// SIMATIC S7-200 SMART project (STEP 7-Micro/WIN SMART), CPU SR20

SYMBOL_TABLE 表格 1
罗茨清洗定时器          T37
螺杆清洗定时器          T38
吹扫定时器            T39
开机吹扫定时器          T41
开机吹扫定时器2         T42
吹扫定时器2           T43
螺杆清洗定时器2         T44
电流保护延时           T40
延时定时器            T55
流量开关定时器          T56
延时触发             V2.0
DCS_启停指令         VW1106   // 1启动、2停机、3复位、4急停
END_SYMBOL_TABLE

SYMBOL_TABLE 系统符号
Always_On        SM0.0    // 始终接通
First_Scan_On    SM0.1    // 仅在第一个扫描周期时接通
END_SYMBOL_TABLE

SYMBOL_TABLE IO过度V10_30
急停_远程            V10.0    // V10~V30
急停_本地            V10.1    // V10~V30
急停标志位            V10.2    // V10~V30
复位_远程            V10.3    // V10~V30
复位_本地            V10.4    // V10~V30
复位标志位            V10.5    // V10~V30
启动_远程            V10.6    // V10~V30
启动_本地            V10.7    // V10~V30
启动标志位            V11.0    // V10~V30
停机_远程            V11.1    // V10~V30
停机_本地            V11.2    // V10~V30
停机标志位            V11.3    // V10~V30
本地_远程            V11.4    // V10~V30
手动_自动            V11.5    // V10~V30
螺杆泵过载_1          V11.6    // V10~V30
螺杆泵过载_2          V11.7    // V10~V30
螺杆泵过载_3          V12.0    // V10~V30
罗茨泵过载_1          V12.1    // V10~V30
罗茨泵过载_2          V12.2    // V10~V30
罗茨泵过载_3          V12.3    // V10~V30
液环泵过载_1          V12.4    // V10~V30
液环泵过载_2          V12.5    // V10~V30
液环泵过载_3          V12.6    // V10~V30
罗茨冷却风机过载_1       V12.7    // V10~V30
罗茨冷却风机过载_2       V13.0    // V10~V30
罗茨冷却风机过载_3       V13.1    // V10~V30
螺杆冷却风机过载_1       V13.2    // V10~V30
螺杆冷却风机过载_2       V13.3    // V10~V30
螺杆冷却风机过载_3       V13.4    // V10~V30
螺杆变频器故障_1        V13.5    // V10~V30
螺杆变频器故障_2        V13.6    // V10~V30
螺杆变频器故障_3        V13.7    // V10~V30
罗茨变频器故障_1        V14.0    // V10~V30
罗茨变频器故障_2        V14.1    // V10~V30
罗茨变频器故障_3        V14.2    // V10~V30
液环软起动故障_1        V14.3    // V10~V30
液环软起动故障_2        V14.4    // V10~V30
液环软起动故障_3        V14.5    // V10~V30
螺杆流量开关_1         V14.6    // V10~V30
螺杆流量开关_2         V14.7    // V10~V30
螺杆流量开关_3         V15.0    // V10~V30
罗茨流量开关_1         V15.1    // V10~V30
罗茨流量开关_2         V15.2    // V10~V30
罗茨流量开关_3         V15.3    // V10~V30
液环流量开关_1         V15.4    // V10~V30
液环流量开关_2         V15.5    // V10~V30
液环流量开关_3         V15.6    // V10~V30
液位开关_1           V15.7    // V10~V30
液位开关_2           V16.0    // V10~V30
液位开关_3           V16.1    // V10~V30
氮封高压开关           V16.2    // V10~V30
氮封低压开关           V16.3    // V10~V30
真空高压开关           V16.4    // V10~V30
真空低压开关           V16.5    // V10~V30
螺杆泵手动_1          V16.6    // V10~V30
螺杆泵手动_2          V16.7    // V10~V30
螺杆泵手动_3          V17.0    // V10~V30
罗茨泵手动_1          V17.1    // V10~V30
罗茨泵手动_2          V17.2    // V10~V30
罗茨泵手动_3          V17.3    // V10~V30
液环泵手动_1          V17.4    // V10~V30
液环泵手动_2          V17.5    // V10~V30
液环泵手动_3          V17.6    // V10~V30
入口阀手动_1          V17.7    // V10~V30
入口阀手动_2          V18.0    // V10~V30
入口阀手动_3          V18.1    // V10~V30
罗茨清洗阀手动          V18.2    // V10~V30
螺杆清洗阀手动          V18.3    // V10~V30
在线清洗阀手动          V18.4    // V10~V30
吹扫阀手动_1          V18.5    // V10~V30
吹扫阀手动_2          V18.6    // V10~V30
吹扫阀手动_3          V18.7    // V10~V30
进水阀手动_1          V19.0    // V10~V30
进水阀手动_2          V19.1    // V10~V30
进水阀手动_3          V19.2    // V10~V30
排污阀手动_1          V19.3    // V10~V30
排污阀手动_2          V19.4    // V10~V30
排污阀手动_3          V19.5    // V10~V30
螺杆1运行时间清零        V19.6    // V10~V30
螺杆2运行时间清零        V19.7    // V10~V30
故障蜂鸣器            V20.0    // V10~V30
停机指示灯            V20.1    // V10~V30
运行指示灯            V20.2    // V10~V30
清洗吹扫指示灯          V20.3    // V10~V30
螺杆泵_1            V20.4    // V10~V30
螺杆泵_2            V20.5    // V10~V30
螺杆泵_3            V20.6    // V10~V30
罗茨泵_1            V20.7    // V10~V30
罗茨泵_2            V21.0    // V10~V30
罗茨泵_3            V21.1    // V10~V30
液环泵_1            V21.2    // V10~V30
液环泵_2            V21.3    // V10~V30
液环泵_3            V21.4    // V10~V30
入口阀_1            V21.5    // V10~V30
入口阀_2            V21.6    // V10~V30
入口阀_3            V21.7    // V10~V30
罗茨清洗阀            V22.0    // V10~V30
螺杆清洗阀1           V22.1    // V10~V30
在线清洗阀            V22.2    // V10~V30
吹扫阀_1            V22.3    // V10~V30
吹扫阀_2            V22.4    // V10~V30
吹扫阀_3            V22.5    // V10~V30
进水阀_1            V22.6    // V10~V30
进水阀_2            V22.7    // V10~V30
进水阀_3            V23.0    // V10~V30
排污阀_1            V23.1    // V10~V30
排污阀_2            V23.2    // V10~V30
排污阀_3            V23.3    // V10~V30
手动标志位            V23.4    // V10~V30
自动标志位            V23.5    // V10~V30
本地标志位            V23.6    // V10~V30
远程标志位            V23.7    // V10~V30
手动控制_一键复位        V24.0    // V10~V30
故障报警_复位_HMI      V24.1    // HMI指令
入口阀1_开到位         V24.2
入口阀1_关到位         V24.3
入口阀2_开到位         V24.4
入口阀2_关到位         V24.5
螺杆清洗阀2           V24.6
螺杆2清洗阀手动         V24.7
启动_自动_HMI        V25.0    // HMI指令
停机_自动_HMI        V25.1    // HMI指令
手动_自动_HMI        V25.2    // HMI指令
本地_远程_HMI        V25.3    // HMI指令
END_SYMBOL_TABLE

SYMBOL_TABLE ABB_MODUBS
主站完成位            M10.0    // M0~M31
开始轮询             M10.1    // M0~M31
通讯完成位_1          M10.2    // M0~M31
通讯完成位_2          M10.3    // M0~M31
通讯完成位_3          M10.4    // M0~M31
通讯完成位_4          M10.5    // M0~M31
通讯完成位_5          M10.6    // M0~M31
通讯完成位_6          M10.7    // M0~M31
主站_校验            MB4      // 0（无奇偶校验）、1（奇校验）和 2（偶校验）。
主站_端口            MB5      // 0 = CPU 中集成的 RS-485，1 = 可选 CM01 信号板上的 RS-485 或 RS-232
轮询步骤             MB8      // M0~M31
主站故障             MB15     // M0~M31
通讯故障_1           MB16     // M0~M31
通讯故障_2           MB17     // M0~M31
通讯故障_3           MB18     // M0~M31
通讯故障_4           MB19     // M0~M31
通讯故障_5           MB20     // M0~M31
通讯故障_6           MB21     // M0~M31
主站_波特率           MD0      // M0~M31
主站_超时            MW6      // M0~M31
频率写入_1           VB104    // VW100~VW200
频率写入_2           VB110    // VW100~VW200
频率写入_3           VB116    // VW100~VW200
频率读取_1           VW100    // VW100~VW200
电流读取_1           VW102    // VW100~VW200
频率读取_2           VW106    // VW100~VW200
电流读取_2           VW108    // VW100~VW200
频率读取_3           VW112    // VW100~VW200
电流读取_3           VW114    // VW100~VW200
频率显示_1           VW150    // VW100~VW200
电流显示_1           VW152    // VW100~VW200
频率显示_2           VW154    // VW100~VW200
电流显示_2           VW156    // VW100~VW200
频率显示_3           VW158    // VW100~VW200
电流显示_3           VW160    // VW100~VW200
END_SYMBOL_TABLE

SYMBOL_TABLE 故障VW218_222
系统1故障            V217.3
系统2故障            V217.4
A类故障             V217.5
B类故障             V217.6
C类故障             V217.7
A_急停_故障          V218.0
A_螺杆流量开关_故障      V218.1   // VW218-VW222
A_螺杆过载_故障        V218.2   // VW218-VW222
A_氮封低压急停_故障      V218.3   // VW218-VW222
A_螺杆温度急停_故障1     V218.4   // VW218-VW222
A_螺杆变频器_故障1      V218.5   // VW218-VW222
A_螺杆变频器_故障2      V218.6   // VW218-VW222
A_螺杆温度急停_故障2     V218.7   // VW218-VW222
预留_A类故障_3        V219.0   // VW218-VW222
预留_A类故障_4        V219.1   // VW218-VW222
预留_A类故障_5        V219.2   // VW218-VW222
预留_A类故障_6        V219.3   // VW218-VW222
预留_A类故障_7        V219.4   // VW218-VW222
预留_A类故障_8        V219.5   // VW218-VW222
预留_A类故障_9        V219.6   // VW218-VW222
预留_A类故障_10       V219.7   // VW218-VW222
B_罗茨过载1_故障       V220.0   // VW218-VW222
B_罗茨1温度停机_故障     V220.1   // VW218-VW222
B_罗茨过载2_故障       V220.2   // VW218-VW222
B_罗茨2温度停机_故障     V220.3   // VW218-VW222
B_罗茨变频器1_故障      V220.4   // VW218-VW222
B_罗茨变频器2_故障      V220.5   // VW218-VW222
B_罗茨变频器3_故障      V220.6   // VW218-VW222
预留_B类故障_1        V220.7   // VW218-VW222
预留_B类故障_2        V221.0   // VW218-VW222
预留_B类故障_3        V221.1   // VW218-VW222
预留_B类故障_4        V221.2   // VW218-VW222
预留_B类故障_5        V221.3   // VW218-VW222
预留_B类故障_6        V221.4   // VW218-VW222
预留_B类故障_7        V221.5   // VW218-VW222
预留_B类故障_8        V221.6   // VW218-VW222
预留_B类故障_9        V221.7   // VW218-VW222
C_罗茨流量开关_故障      V222.0   // VW218-VW222
C_螺杆温度报警_故障1     V222.1   // VW218-VW222
C_氮封高压报警_故障      V222.2   // VW218-VW222
C_液位过高报警_故障      V222.3   // VW218-VW222
C_罗茨温度报警_故障      V222.4   // VW218-VW222
C_螺杆温度报警_故障2     V222.5   // VW218-VW222
预留_C类故障_2        V222.6   // VW218-VW222
预留_C类故障_3        V222.7   // VW218-VW222
预留_C类故障_4        V223.0   // VW218-VW222
预留_C类故障_5        V223.1   // VW218-VW222
预留_C类故障_6        V223.2   // VW218-VW222
预留_C类故障_7        V223.3   // VW218-VW222
预留_C类故障_8        V223.4   // VW218-VW222
预留_C类故障_9        V223.5   // VW218-VW222
预留_C类故障_10       V223.6   // VW218-VW222
预留_C类故障_11       V223.7   // VW218-VW222
END_SYMBOL_TABLE

SYMBOL_TABLE 参数设置VW1000_1148
罗茨_温度报警_设置       VD1000   // VW1000~VW1148
罗茨_温度停机_设置       VD1004   // VW1000~VW1148
液位_过高报警_设置       VD1008   // VW1000~VW1148
螺杆_温度报警_设置       VD1012   // VW1000~VW1148
螺杆_温度停机_设置       VD1016   // VW1000~VW1148
电流_保护_设置         VD1020   // VW1000~VW1148
电流_恢复_设置         VD1024   // VW1000~VW1148
液位_保护_设置         VD1028   // VW1000~VW1148
液位_恢复_设置         VD1032   // VW1000~VW1148
液位_变送器上限_设置      VD1036   // VW1000~VW1148
螺杆温度_变送器上限_设     VD1040   // VW1000~VW1148
电流_变送器上限_设置      VD1044   // VW1000~VW1148
罗茨1温度_变送器上限_设    VD1048   // VW1000~VW1148
罗茨2温度_变送器上限_设    VD1052   // VW1000~VW1148
罗茨1启动真空设定        VD1056   // VW1000~VW1148
罗茨1停机真空设定        VD1060   // VW1000~VW1148
罗茨2启动真空设定        VD1064   // VW1000~VW1148
罗茨2停机真空设定        VD1068   // VW1000~VW1148
真空_变送器上限_设定      VD1072   // VW1000~VW1148
氮气_变送器上限_设定      VD1076   // VW1000~VW1148
氮气_低压急停_设定       VD1080   // VW1000~VW1148
氮气_低压报警_设定       VD1084   // VW1000~VW1148
目标真空度_设定         VD1088   // VW1000~VW1148
                 VD1092   // VW1000~VW1148
                 VD1096   // VW1000~VW1148
DCS_校验_设置        VD1144   // VW1000~VW1148
罗茨_清洗时间_设置       VW1100   // VW1000~VW1148
螺杆_清洗时间_设置       VW1102   // VW1000~VW1148
吹扫_时间_设置         VW1104   // VW1000~VW1148
螺杆手动频率_设置        VW1108   // VW1000~VW1148
罗茨1手动频率_设置       VW1110   // VW1000~VW1148
罗茨2手动频率_设置       VW1112   // VW1000~VW1148
螺杆清洗频率_设置        VW1114   // VW1000~VW1148
螺杆2手动频率_设置       VW1116   // VW1000~VW1148
螺杆2清洗频率_设置       VW1118   // VW1000~VW1148
开机吹扫_时间_设置       VW1120   // VW1000~VW1148
电流过载_预防_设置       VW1122   // VW1000~VW1148
                 VW1124   // VW1000~VW1148
                 VW1126   // VW1000~VW1148
                 VW1128   // VW1000~VW1148
                 VW1130   // VW1000~VW1148
                 VW1132   // VW1000~VW1148
                 VW1134   // VW1000~VW1148
                 VW1136   // VW1000~VW1148
                 VW1138   // VW1000~VW1148
DCS_地址_设置        VW1140   // VW1000~VW1148
DCS_波特率_设置       VW1142   // VW1000~VW1148
                 VW1148   // VW1000~VW1148
                          // VW1000~VW1148
END_SYMBOL_TABLE

SYMBOL_TABLE 参数显示
螺杆温度值1           VD1154
罗茨液位值            VD1158
螺杆液位值            VD1162
螺杆电流值            VD1166
机组真空度            VD1170
罗茨温度值            VD1178
绝对真空显示           VD1182
自动步骤1            VW1202
自动步骤2            VW1204
开机吹扫_时间_显示       VW1206
螺杆_清洗时间_显示       VW1208
罗茨_清洗时间_显示       VW1210
吹扫时间_显示          VW1212
螺杆_频率_显示         VW1214
螺杆_电流_显示         VW1216
罗茨1_频率_显示        VW1218
罗茨1_电流_显示        VW1220
罗茨2_频率_显示        VW1222
罗茨2_电流_显示        VW1224
螺杆1运行时间_秒        VW1226
螺杆1运行时间_分        VW1228
螺杆1运行时间_时        VW1230
螺杆2运行时间_秒        VW1232
螺杆2运行时间_分        VW1234
螺杆2运行时间_时        VW1236
螺杆温度值2           VD1186
螺杆温度值3           VD1190
入口温度1            VD1194
入口温度2            VD1198
螺杆2_频率_显示        VW1238
螺杆2_电流_显示        VW1240
END_SYMBOL_TABLE

SYMBOL_TABLE 变送器VD30_96
真空变送器            VW30     // VD30~VD96
螺杆温度变送器_1        VW32     // VD30~VD96
螺杆温度变送器_2        VW34     // VD30~VD96
螺杆温度变送器_3        VW36     // VD30~VD96
罗茨温度变送器_1        VW38     // VD30~VD96
罗茨温度变送器_2        VW40     // VD30~VD96
罗茨温度变送器_3        VW42     // VD30~VD96
液环温度变送器_1        VW44     // VD30~VD96
液环温度变送器_2        VW46     // VD30~VD96
液环温度变送器_3        VW48     // VD30~VD96
入口温度变送器1         VW50     // VD30~VD96
液位变送器            VW52     // VD30~VD96
前端液位变送器          VW54     // VD30~VD96
后端液位变送器          VW56     // VD30~VD96
螺杆电流变送器          VW58     // VD30~VD96
入口温度变送器2         VW60     // VD30~VD96
END_SYMBOL_TABLE

SYMBOL_TABLE 辅助点表
急停_远程_使能         V300.0
急停_本地_使能         V300.1
急停标志位_使能         V300.2
复位_远程_使能         V300.3
复位_本地_使能         V300.4
复位标志位_使能         V300.5
启动_远程_使能         V300.6
启动_本地_使能         V300.7
启动标志位_使能         V301.0
停机_远程_使能         V301.1
停机_本地_使能         V301.2
停机标志位_使能         V301.3
本地_远程_使能         V301.4
手动_自动_使能         V301.5
螺杆泵过载_1_使能       V301.6
螺杆泵过载_2_使能       V301.7
螺杆泵过载_3_使能       V302.0
罗茨泵过载_1_使能       V302.1
罗茨泵过载_2_使能       V302.2
罗茨泵过载_3_使能       V302.3
液环泵过载_1_使能       V302.4
液环泵过载_2_使能       V302.5
液环泵过载_3_使能       V302.6
罗茨冷却风机过载_1_使能    V302.7
罗茨冷却风机过载_2_使能    V303.0
罗茨冷却风机过载_3_使能    V303.1
螺杆冷却风机过载_1_使能    V303.2
螺杆冷却风机过载_2_使能    V303.3
螺杆冷却风机过载_3_使能    V303.4
螺杆变频器故障_1_使能     V303.5
螺杆变频器故障_2_使能     V303.6
螺杆变频器故障_3_使能     V303.7
罗茨变频器故障_1_使能     V304.0
罗茨变频器故障_2_使能     V304.1
罗茨变频器故障_3_使能     V304.2
液环软起动故障_1_使能     V304.3
液环软起动故障_2_使能     V304.4
液环软起动故障_3_使能     V304.5
螺杆流量开关_1_使能      V304.6
螺杆流量开关_2_使能      V304.7
螺杆流量开关_3_使能      V305.0
罗茨流量开关_1_使能      V305.1
罗茨流量开关_2_使能      V305.2
罗茨流量开关_3_使能      V305.3
液环流量开关_1_使能      V305.4
液环流量开关_2_使能      V305.5
液环流量开关_3_使能      V305.6
液位开关_1_使能        V305.7
液位开关_2_使能        V306.0
液位开关_3_使能        V306.1
氮封高压开关_使能        V306.2
氮封低压开关_使能        V306.3
真空高压开关_使能        V306.4
真空低压开关_使能        V306.5
螺杆泵手动_1_使能       V306.6
螺杆泵手动_2_使能       V306.7
螺杆泵手动_3_使能       V307.0
罗茨泵手动_1_使能       V307.1
罗茨泵手动_2_使能       V307.2
罗茨泵手动_3_使能       V307.3
液环泵手动_1_使能       V307.4
液环泵手动_2_使能       V307.5
液环泵手动_3_使能       V307.6
入口阀手动_1_使能       V307.7
入口阀手动_2_使能       V308.0
入口阀手动_3_使能       V308.1
罗茨清洗阀手动_使能       V308.2
螺杆1清洗阀手动_使能      V308.3
在线清洗阀手动_使能       V308.4
吹扫阀手动_1_使能       V308.5
吹扫阀手动_2_使能       V308.6
吹扫阀手动_3_使能       V308.7
进水阀手动_1_使能       V309.0
进水阀手动_2_使能       V309.1
进水阀手动_3_使能       V309.2
排污阀手动_1_使能       V309.3
排污阀手动_2_使能       V309.4
排污阀手动_3_使能       V309.5
螺杆1运行时间清零_使能     V309.6
螺杆2运行时间清零_使能     V309.7
故障蜂鸣器_使能         V310.0
停机指示灯_使能         V310.1
运行指示灯_使能         V310.2
清洗吹扫指示灯_使能       V310.3
螺杆泵_1_使能         V310.4
螺杆泵_2_使能         V310.5
螺杆泵_3_使能         V310.6
罗茨泵_1_使能         V310.7
罗茨泵_2_使能         V311.0
罗茨泵_3_使能         V311.1
液环泵_1_使能         V311.2
液环泵_2_使能         V311.3
液环泵_3_使能         V311.4
入口阀_1_使能         V311.5
入口阀_2_使能         V311.6
入口阀_3_使能         V311.7
罗茨清洗阀_使能         V312.0
螺杆清洗阀1_使能        V312.1
在线清洗阀_使能         V312.2
吹扫阀_1_使能         V312.3
吹扫阀_2_使能         V312.4
吹扫阀_3_使能         V312.5
进水阀_1_使能         V312.6
进水阀_2_使能         V312.7
进水阀_3_使能         V313.0
排污阀_1_使能         V313.1
排污阀_2_使能         V313.2
排污阀_3_使能         V313.3
手动标志位_使能         V313.4
自动标志位_使能         V313.5
本地标志位_使能         V313.6
远程标志位_使能         V313.7
手动控制_一键复位_使能     V314.0
故障报警_复位_HMI_使能   V314.1
入口阀1_开到位_使能      V314.2
入口阀1_关到位_使能      V314.3
入口阀2_开到位_使能      V314.4
入口阀2_关到位_使能      V314.5
螺杆清洗阀2_使能        V314.6
系统1_使能           V315.0
系统2_使能           V315.1
系统3_使能           V315.2
优先启动机组           V315.3
螺杆2清洗阀手动_使能      V314.7
END_SYMBOL_TABLE

SYMBOL_TABLE 中间变量
开机吹扫_时间_中间值      VW5000
吹扫_时间_中间值        VW5002
螺杆_清洗时间_中间值      VW5004
罗茨_清洗时间_中间值      VW5006
PID_频率1          VW5008
PID_频率2          VW5010
END_SYMBOL_TABLE

SYMBOL_TABLE PID数据
PID故障1           VB5200
PID故障2           VB5201
END_SYMBOL_TABLE

ORGANIZATION_BLOCK MAIN:OB1
TITLE=程序注释
BEGIN
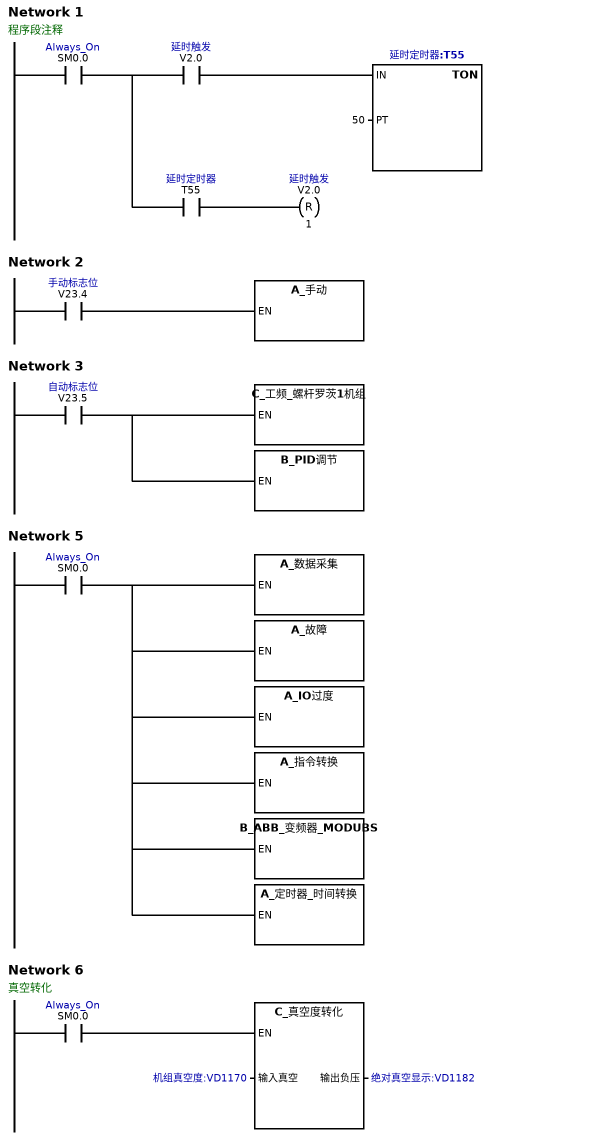
Network 1
// 程序段注释
LD     Always_On:SM0.0
LPS
A      延时触发:V2.0
TON    延时定时器:T55, 50
LPP
A      延时定时器:T55
R      延时触发:V2.0, 1
Network 2
LD     手动标志位:V23.4
CALL   A_手动:SBR0
Network 3
LD     自动标志位:V23.5
CALL   C_工频_螺杆罗茨1机组:SBR1
CALL   B_PID调节:SBR22
Network 5
LD     Always_On:SM0.0
CALL   A_数据采集:SBR2
CALL   A_故障:SBR3
CALL   A_IO过度:SBR5
CALL   A_指令转换:SBR11
CALL   B_ABB_变频器_MODUBS:SBR7
CALL   A_定时器_时间转换:SBR21
Network 6
// 真空转化
LD     Always_On:SM0.0
CALL   C_真空度转化:SBR12, 机组真空度:VD1170, 绝对真空显示:VD1182
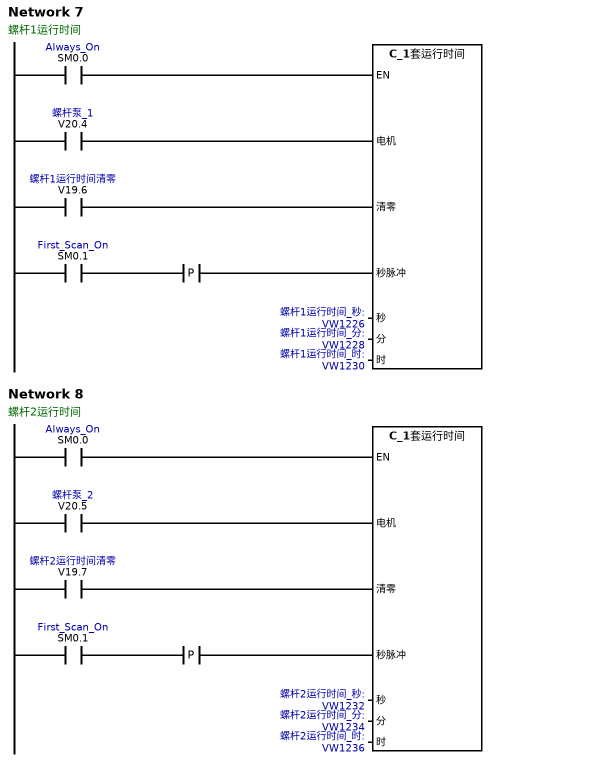
Network 7
// 螺杆1运行时间
LD     Always_On:SM0.0
=      L60.0
LD     螺杆泵_1:V20.4
=      L63.7
LD     螺杆1运行时间清零:V19.6
=      L63.6
LD     First_Scan_On:SM0.1
EU
=      L63.5
LD     L60.0
CALL   C_1套运行时间:SBR13, L63.7, L63.6, L63.5, 螺杆1运行时间_秒:VW1226, 螺杆1运行时间_分:VW1228, 螺杆1运行时间_时:VW1230
Network 8
// 螺杆2运行时间
LD     Always_On:SM0.0
=      L60.0
LD     螺杆泵_2:V20.5
=      L63.7
LD     螺杆2运行时间清零:V19.7
=      L63.6
LD     First_Scan_On:SM0.1
EU
=      L63.5
LD     L60.0
CALL   C_1套运行时间:SBR13, L63.7, L63.6, L63.5, 螺杆2运行时间_秒:VW1232, 螺杆2运行时间_分:VW1234, 螺杆2运行时间_时:VW1236
END_ORGANIZATION_BLOCK

SUBROUTINE_BLOCK A_手动:SBR0
TITLE=子程序注释
BEGIN
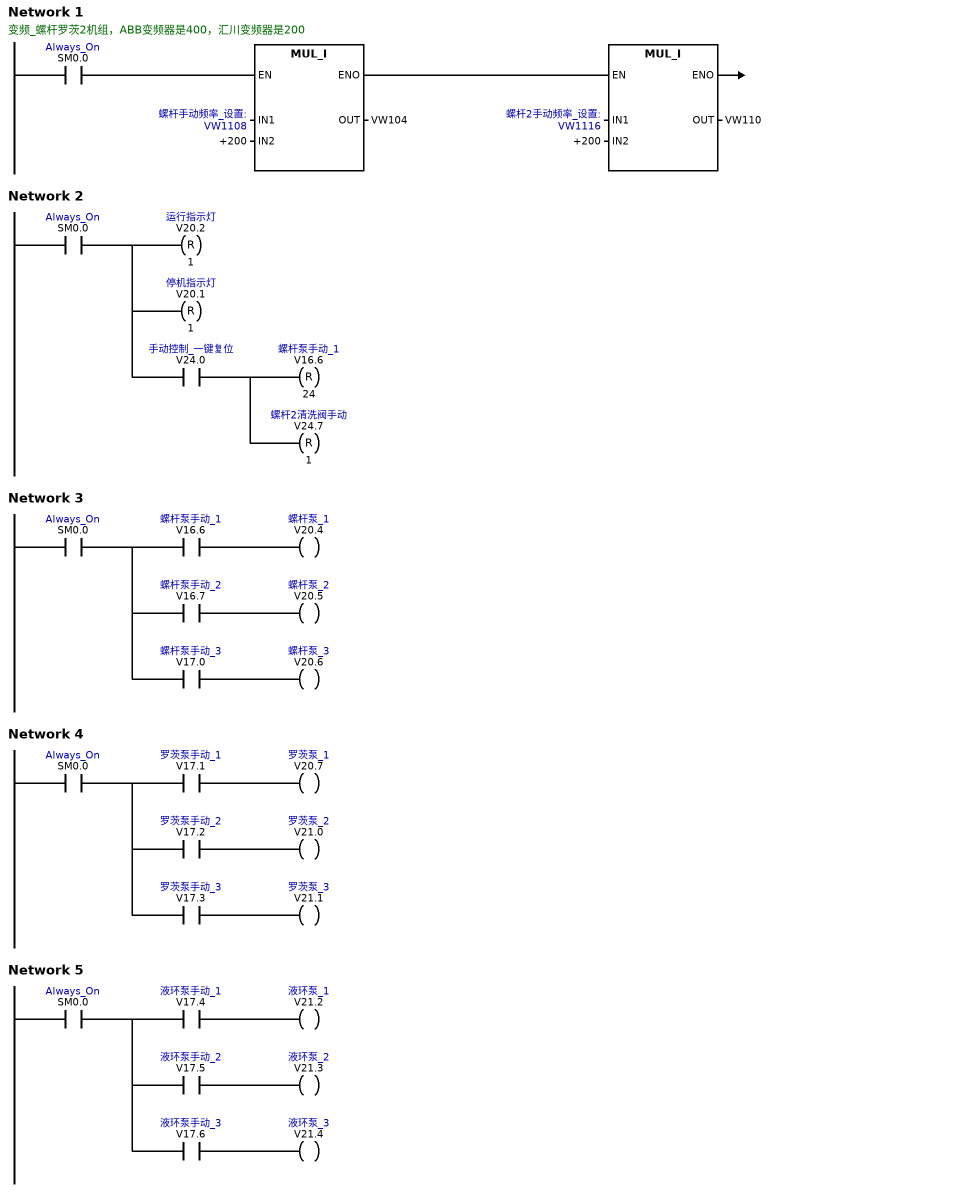
Network 1
// 变频_螺杆罗茨2机组，ABB变频器是400，汇川变频器是200
LD     Always_On:SM0.0
MOVW   螺杆手动频率_设置:VW1108, VW104
AENO
*I     +200, VW104
AENO
MOVW   螺杆2手动频率_设置:VW1116, VW110
*I     +200, VW110
Network 2
LD     Always_On:SM0.0
R      运行指示灯:V20.2, 1
R      停机指示灯:V20.1, 1
A      手动控制_一键复位:V24.0
R      螺杆泵手动_1:V16.6, 24
R      螺杆2清洗阀手动:V24.7, 1
Network 3
LD     Always_On:SM0.0
LPS
A      螺杆泵手动_1:V16.6
=      螺杆泵_1:V20.4
LRD
A      螺杆泵手动_2:V16.7
=      螺杆泵_2:V20.5
LPP
A      螺杆泵手动_3:V17.0
=      螺杆泵_3:V20.6
Network 4
LD     Always_On:SM0.0
LPS
A      罗茨泵手动_1:V17.1
=      罗茨泵_1:V20.7
LRD
A      罗茨泵手动_2:V17.2
=      罗茨泵_2:V21.0
LPP
A      罗茨泵手动_3:V17.3
=      罗茨泵_3:V21.1
Network 5
LD     Always_On:SM0.0
LPS
A      液环泵手动_1:V17.4
=      液环泵_1:V21.2
LRD
A      液环泵手动_2:V17.5
=      液环泵_2:V21.3
LPP
A      液环泵手动_3:V17.6
=      液环泵_3:V21.4
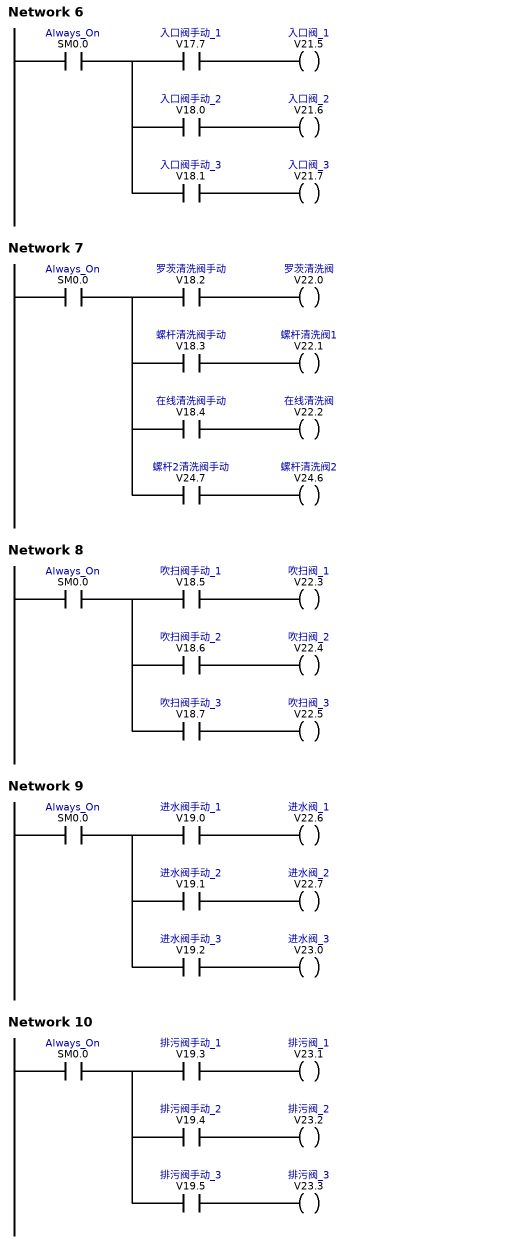
Network 6
LD     Always_On:SM0.0
LPS
A      入口阀手动_1:V17.7
=      入口阀_1:V21.5
LRD
A      入口阀手动_2:V18.0
=      入口阀_2:V21.6
LPP
A      入口阀手动_3:V18.1
=      入口阀_3:V21.7
Network 7
LD     Always_On:SM0.0
LPS
A      罗茨清洗阀手动:V18.2
=      罗茨清洗阀:V22.0
LRD
A      螺杆清洗阀手动:V18.3
=      螺杆清洗阀1:V22.1
LRD
A      在线清洗阀手动:V18.4
=      在线清洗阀:V22.2
LPP
A      螺杆2清洗阀手动:V24.7
=      螺杆清洗阀2:V24.6
Network 8
LD     Always_On:SM0.0
LPS
A      吹扫阀手动_1:V18.5
=      吹扫阀_1:V22.3
LRD
A      吹扫阀手动_2:V18.6
=      吹扫阀_2:V22.4
LPP
A      吹扫阀手动_3:V18.7
=      吹扫阀_3:V22.5
Network 9
LD     Always_On:SM0.0
LPS
A      进水阀手动_1:V19.0
=      进水阀_1:V22.6
LRD
A      进水阀手动_2:V19.1
=      进水阀_2:V22.7
LPP
A      进水阀手动_3:V19.2
=      进水阀_3:V23.0
Network 10
LD     Always_On:SM0.0
LPS
A      排污阀手动_1:V19.3
=      排污阀_1:V23.1
LRD
A      排污阀手动_2:V19.4
=      排污阀_2:V23.2
LPP
A      排污阀手动_3:V19.5
=      排污阀_3:V23.3
END_SUBROUTINE_BLOCK

SUBROUTINE_BLOCK C_工频_螺杆罗茨1机组:SBR1
TITLE=子程序注释
BEGIN
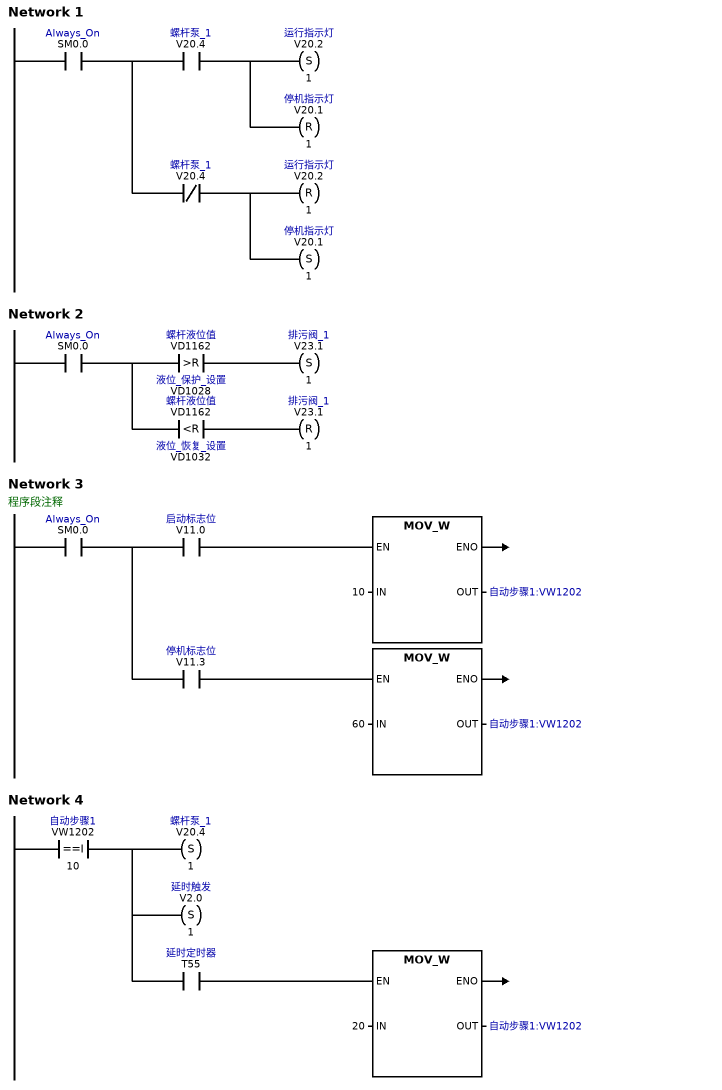
Network 1
LD     Always_On:SM0.0
LPS
A      螺杆泵_1:V20.4
S      运行指示灯:V20.2, 1
R      停机指示灯:V20.1, 1
LPP
AN     螺杆泵_1:V20.4
R      运行指示灯:V20.2, 1
S      停机指示灯:V20.1, 1
Network 2
LD     Always_On:SM0.0
LPS
AR>    螺杆液位值:VD1162, 液位_保护_设置:VD1028
S      排污阀_1:V23.1, 1
LPP
AR<    螺杆液位值:VD1162, 液位_恢复_设置:VD1032
R      排污阀_1:V23.1, 1
Network 3
// 程序段注释
LD     Always_On:SM0.0
LPS
A      启动标志位:V11.0
MOVW   10, 自动步骤1:VW1202
LPP
A      停机标志位:V11.3
MOVW   60, 自动步骤1:VW1202
Network 4
LDW=   自动步骤1:VW1202, 10
S      螺杆泵_1:V20.4, 1
S      延时触发:V2.0, 1
A      延时定时器:T55
MOVW   20, 自动步骤1:VW1202
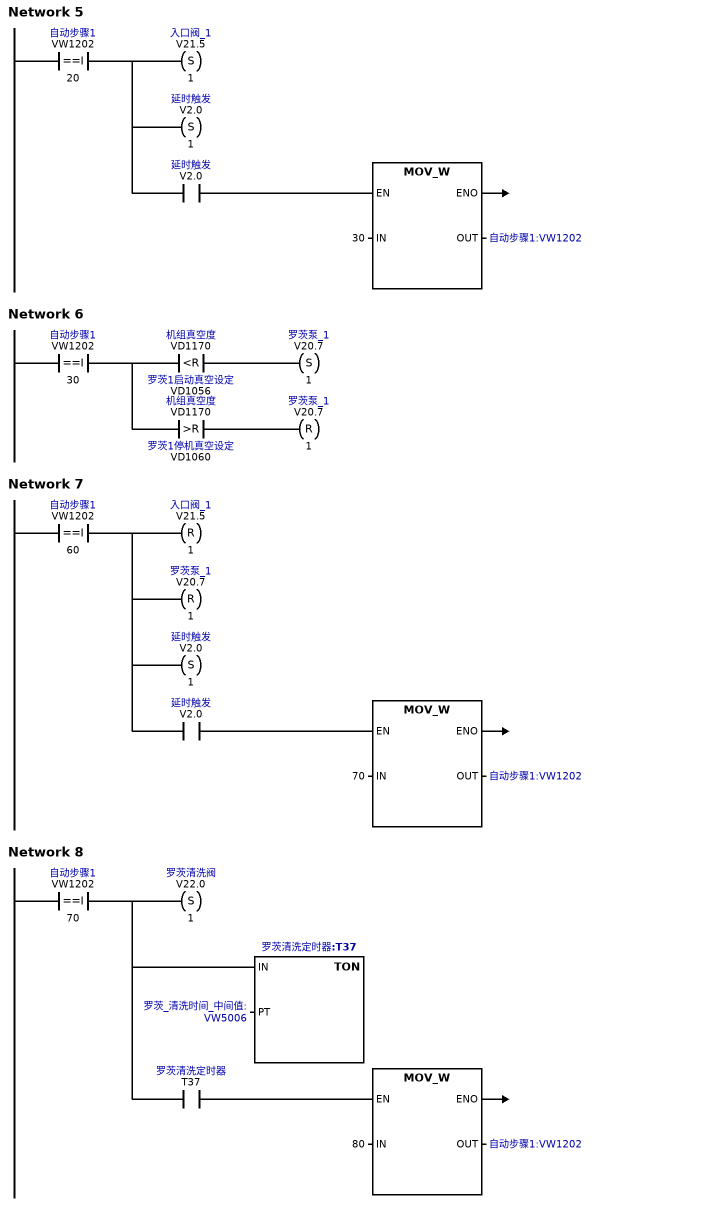
Network 5
LDW=   自动步骤1:VW1202, 20
S      入口阀_1:V21.5, 1
S      延时触发:V2.0, 1
A      延时触发:V2.0
MOVW   30, 自动步骤1:VW1202
Network 6
LDW=   自动步骤1:VW1202, 30
LPS
AR<    机组真空度:VD1170, 罗茨1启动真空设定:VD1056
S      罗茨泵_1:V20.7, 1
LPP
AR>    机组真空度:VD1170, 罗茨1停机真空设定:VD1060
R      罗茨泵_1:V20.7, 1
Network 7
LDW=   自动步骤1:VW1202, 60
R      入口阀_1:V21.5, 1
R      罗茨泵_1:V20.7, 1
S      延时触发:V2.0, 1
A      延时触发:V2.0
MOVW   70, 自动步骤1:VW1202
Network 8
LDW=   自动步骤1:VW1202, 70
S      罗茨清洗阀:V22.0, 1
TON    罗茨清洗定时器:T37, 罗茨_清洗时间_中间值:VW5006
A      罗茨清洗定时器:T37
MOVW   80, 自动步骤1:VW1202
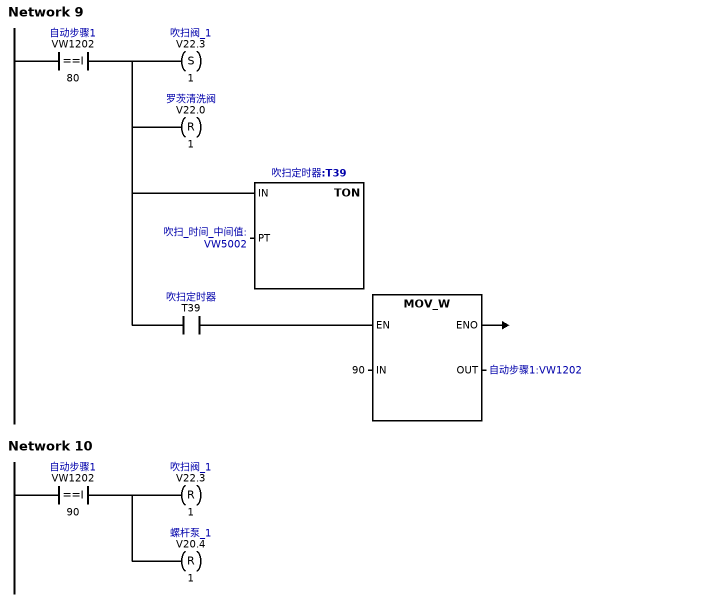
Network 9
LDW=   自动步骤1:VW1202, 80
S      吹扫阀_1:V22.3, 1
R      罗茨清洗阀:V22.0, 1
TON    吹扫定时器:T39, 吹扫_时间_中间值:VW5002
A      吹扫定时器:T39
MOVW   90, 自动步骤1:VW1202
Network 10
LDW=   自动步骤1:VW1202, 90
R      吹扫阀_1:V22.3, 1
R      螺杆泵_1:V20.4, 1
END_SUBROUTINE_BLOCK

SUBROUTINE_BLOCK A_数据采集:SBR2
TITLE=子程序注释
BEGIN
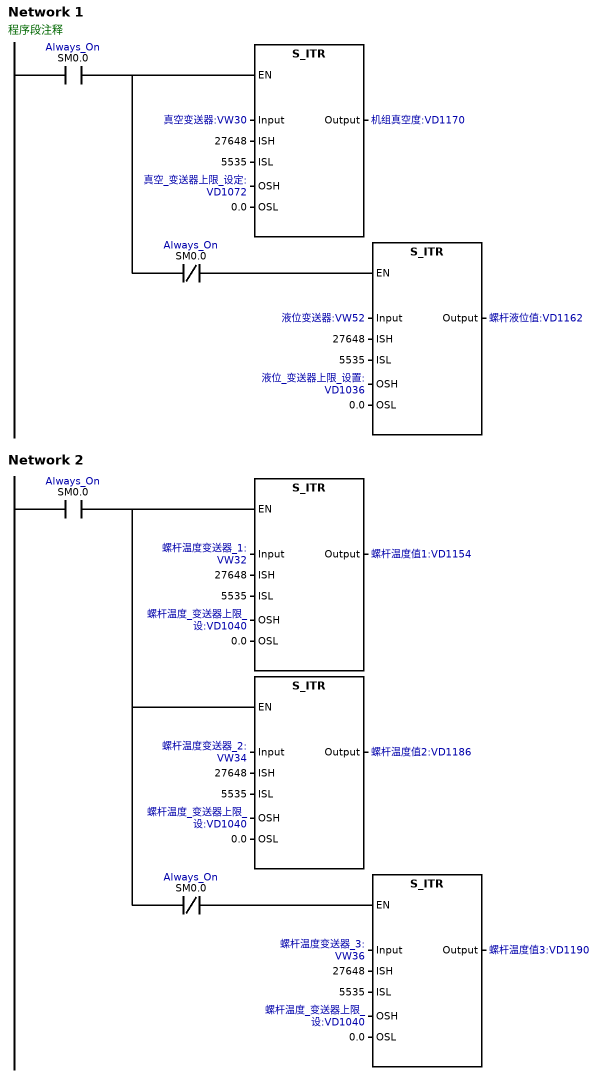
Network 1
// 程序段注释
LD     Always_On:SM0.0
CALL   S_ITR:SBR4, 真空变送器:VW30, 27648, 5535, 真空_变送器上限_设定:VD1072, 0.0, 机组真空度:VD1170
AN     Always_On:SM0.0
CALL   S_ITR:SBR4, 液位变送器:VW52, 27648, 5535, 液位_变送器上限_设置:VD1036, 0.0, 螺杆液位值:VD1162
Network 2
LD     Always_On:SM0.0
CALL   S_ITR:SBR4, 螺杆温度变送器_1:VW32, 27648, 5535, 螺杆温度_变送器上限_设:VD1040, 0.0, 螺杆温度值1:VD1154
CALL   S_ITR:SBR4, 螺杆温度变送器_2:VW34, 27648, 5535, 螺杆温度_变送器上限_设:VD1040, 0.0, 螺杆温度值2:VD1186
AN     Always_On:SM0.0
CALL   S_ITR:SBR4, 螺杆温度变送器_3:VW36, 27648, 5535, 螺杆温度_变送器上限_设:VD1040, 0.0, 螺杆温度值3:VD1190
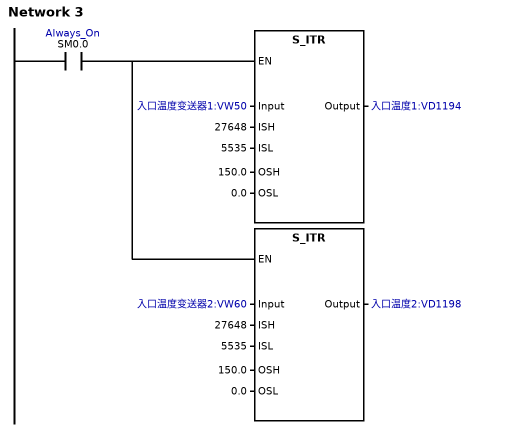
Network 3
LD     Always_On:SM0.0
CALL   S_ITR:SBR4, 入口温度变送器1:VW50, 27648, 5535, 150.0, 0.0, 入口温度1:VD1194
CALL   S_ITR:SBR4, 入口温度变送器2:VW60, 27648, 5535, 150.0, 0.0, 入口温度2:VD1198
END_SUBROUTINE_BLOCK

SUBROUTINE_BLOCK A_故障:SBR3
TITLE=子程序注释
BEGIN
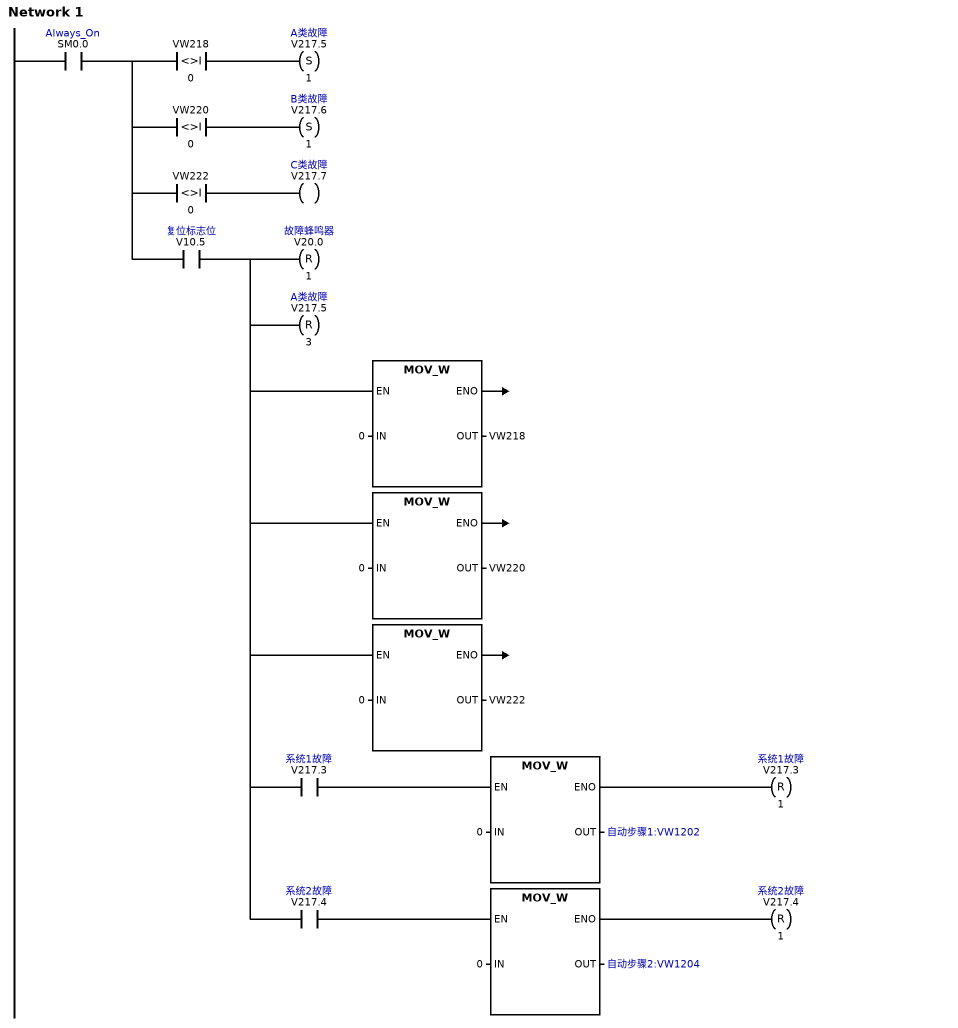
Network 1
LD     Always_On:SM0.0
LPS
AW<>   VW218, 0
S      A类故障:V217.5, 1
LRD
AW<>   VW220, 0
S      B类故障:V217.6, 1
LRD
AW<>   VW222, 0
=      C类故障:V217.7
LPP
A      复位标志位:V10.5
LPS
R      故障蜂鸣器:V20.0, 1
R      A类故障:V217.5, 3
MOVW   0, VW218
MOVW   0, VW220
MOVW   0, VW222
A      系统1故障:V217.3
MOVW   0, 自动步骤1:VW1202
AENO
R      系统1故障:V217.3, 1
LPP
A      系统2故障:V217.4
MOVW   0, 自动步骤2:VW1204
AENO
R      系统2故障:V217.4, 1
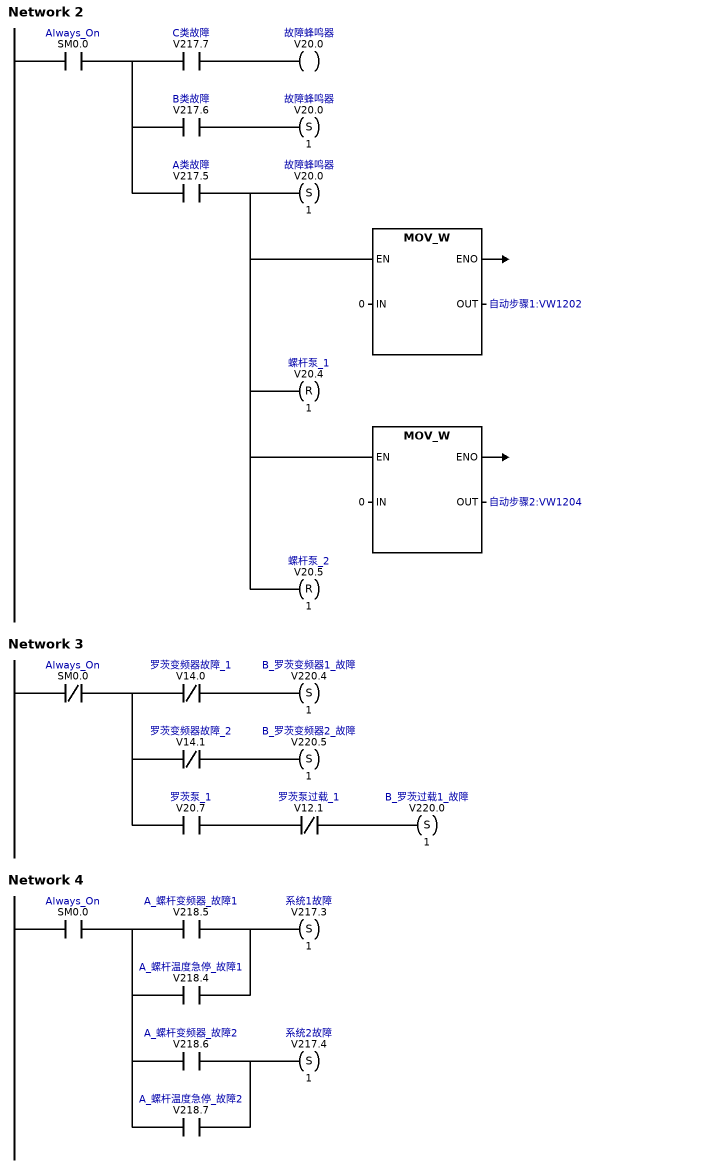
Network 2
LD     Always_On:SM0.0
LPS
A      C类故障:V217.7
=      故障蜂鸣器:V20.0
LRD
A      B类故障:V217.6
S      故障蜂鸣器:V20.0, 1
LPP
A      A类故障:V217.5
S      故障蜂鸣器:V20.0, 1
MOVW   0, 自动步骤1:VW1202
R      螺杆泵_1:V20.4, 1
MOVW   0, 自动步骤2:VW1204
R      螺杆泵_2:V20.5, 1
Network 3
LDN    Always_On:SM0.0
LPS
AN     罗茨变频器故障_1:V14.0
S      B_罗茨变频器1_故障:V220.4, 1
LRD
AN     罗茨变频器故障_2:V14.1
S      B_罗茨变频器2_故障:V220.5, 1
LPP
A      罗茨泵_1:V20.7
AN     罗茨泵过载_1:V12.1
S      B_罗茨过载1_故障:V220.0, 1
Network 4
LD     Always_On:SM0.0
LPS
LD     A_螺杆变频器_故障1:V218.5
O      A_螺杆温度急停_故障1:V218.4
ALD
S      系统1故障:V217.3, 1
LPP
LD     A_螺杆变频器_故障2:V218.6
O      A_螺杆温度急停_故障2:V218.7
ALD
S      系统2故障:V217.4, 1
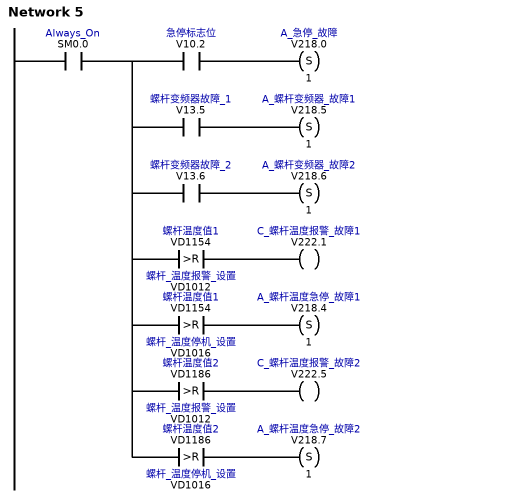
Network 5
LD     Always_On:SM0.0
LPS
A      急停标志位:V10.2
S      A_急停_故障:V218.0, 1
LRD
A      螺杆变频器故障_1:V13.5
S      A_螺杆变频器_故障1:V218.5, 1
LRD
A      螺杆变频器故障_2:V13.6
S      A_螺杆变频器_故障2:V218.6, 1
LRD
AR>    螺杆温度值1:VD1154, 螺杆_温度报警_设置:VD1012
=      C_螺杆温度报警_故障1:V222.1
LRD
AR>    螺杆温度值1:VD1154, 螺杆_温度停机_设置:VD1016
S      A_螺杆温度急停_故障1:V218.4, 1
LRD
AR>    螺杆温度值2:VD1186, 螺杆_温度报警_设置:VD1012
=      C_螺杆温度报警_故障2:V222.5
LPP
AR>    螺杆温度值2:VD1186, 螺杆_温度停机_设置:VD1016
S      A_螺杆温度急停_故障2:V218.7, 1
END_SUBROUTINE_BLOCK

// SBR4: protected block, not included

SUBROUTINE_BLOCK A_IO过度:SBR5
TITLE=DI,DO,AI,AO过渡，占用V10~100
BEGIN
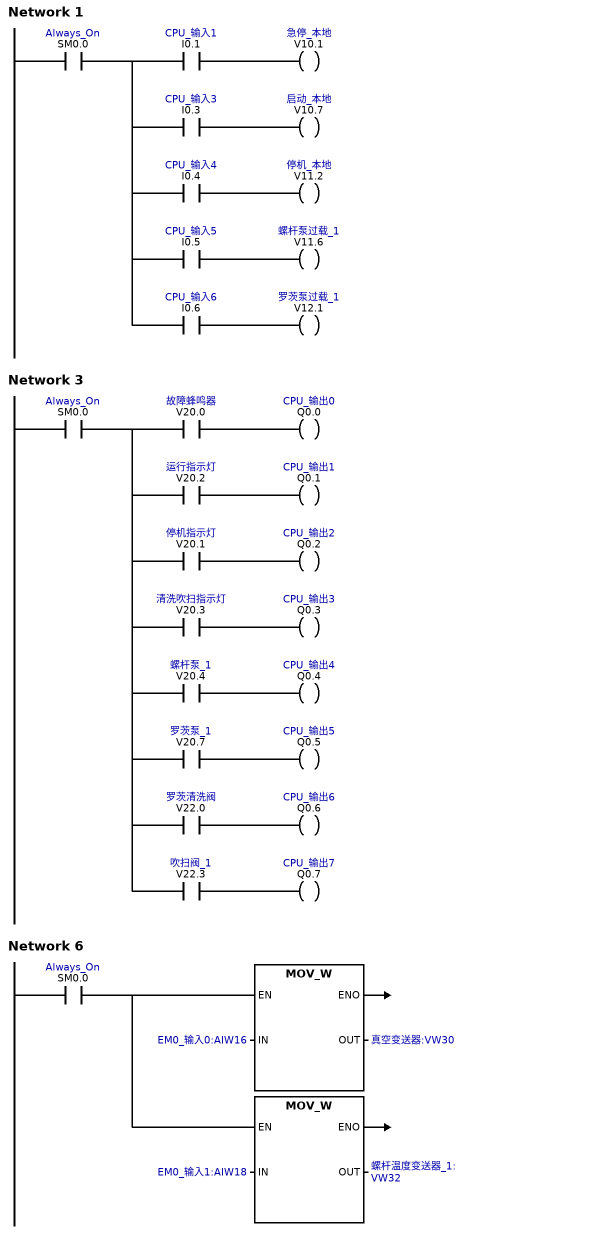
Network 1
LD     Always_On:SM0.0
LPS
A      CPU_输入1:I0.1
=      急停_本地:V10.1
LRD
A      CPU_输入3:I0.3
=      启动_本地:V10.7
LRD
A      CPU_输入4:I0.4
=      停机_本地:V11.2
LRD
A      CPU_输入5:I0.5
=      螺杆泵过载_1:V11.6
LPP
A      CPU_输入6:I0.6
=      罗茨泵过载_1:V12.1
Network 3
LD     Always_On:SM0.0
LPS
A      故障蜂鸣器:V20.0
=      CPU_输出0:Q0.0
LRD
A      运行指示灯:V20.2
=      CPU_输出1:Q0.1
LRD
A      停机指示灯:V20.1
=      CPU_输出2:Q0.2
LRD
A      清洗吹扫指示灯:V20.3
=      CPU_输出3:Q0.3
LRD
A      螺杆泵_1:V20.4
=      CPU_输出4:Q0.4
LRD
A      罗茨泵_1:V20.7
=      CPU_输出5:Q0.5
LRD
A      罗茨清洗阀:V22.0
=      CPU_输出6:Q0.6
LPP
A      吹扫阀_1:V22.3
=      CPU_输出7:Q0.7
Network 6
LD     Always_On:SM0.0
MOVW   EM0_输入0:AIW16, 真空变送器:VW30
MOVW   EM0_输入1:AIW18, 螺杆温度变送器_1:VW32
END_SUBROUTINE_BLOCK

SUBROUTINE_BLOCK C_变频_螺杆罗茨2机组:SBR6
TITLE=子程序注释
BEGIN
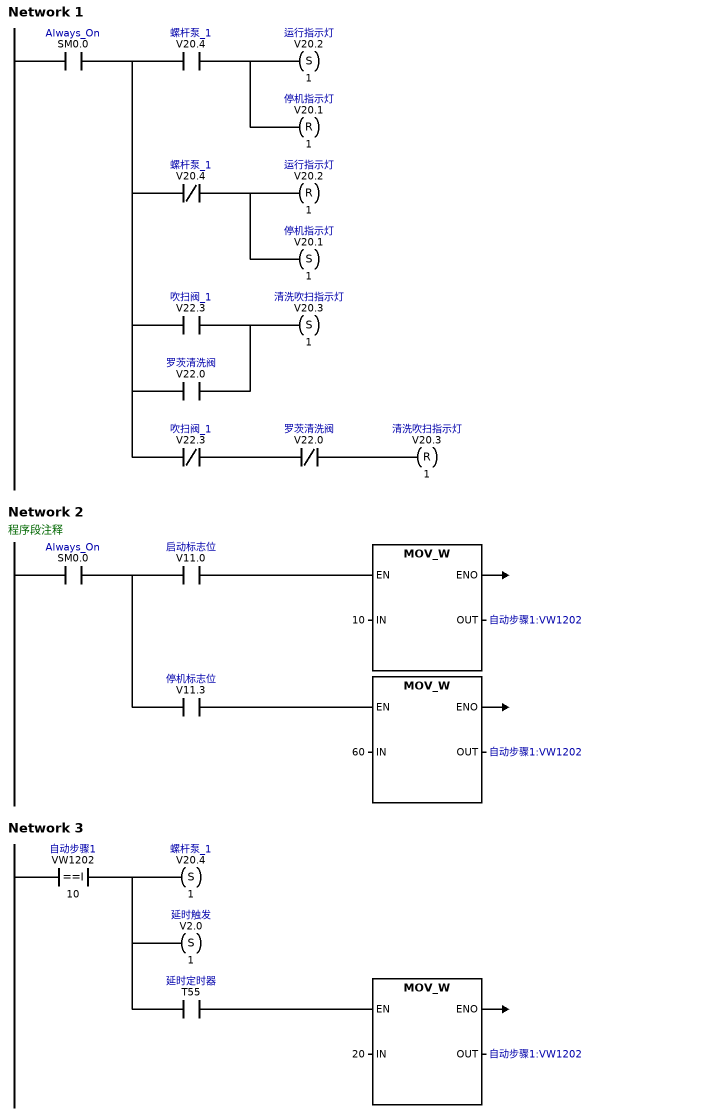
Network 1
LD     Always_On:SM0.0
LPS
A      螺杆泵_1:V20.4
S      运行指示灯:V20.2, 1
R      停机指示灯:V20.1, 1
LRD
AN     螺杆泵_1:V20.4
R      运行指示灯:V20.2, 1
S      停机指示灯:V20.1, 1
LRD
LD     吹扫阀_1:V22.3
O      罗茨清洗阀:V22.0
ALD
S      清洗吹扫指示灯:V20.3, 1
LPP
AN     吹扫阀_1:V22.3
AN     罗茨清洗阀:V22.0
R      清洗吹扫指示灯:V20.3, 1
Network 2
// 程序段注释
LD     Always_On:SM0.0
LPS
A      启动标志位:V11.0
MOVW   10, 自动步骤1:VW1202
LPP
A      停机标志位:V11.3
MOVW   60, 自动步骤1:VW1202
Network 3
LDW=   自动步骤1:VW1202, 10
S      螺杆泵_1:V20.4, 1
S      延时触发:V2.0, 1
A      延时定时器:T55
MOVW   20, 自动步骤1:VW1202
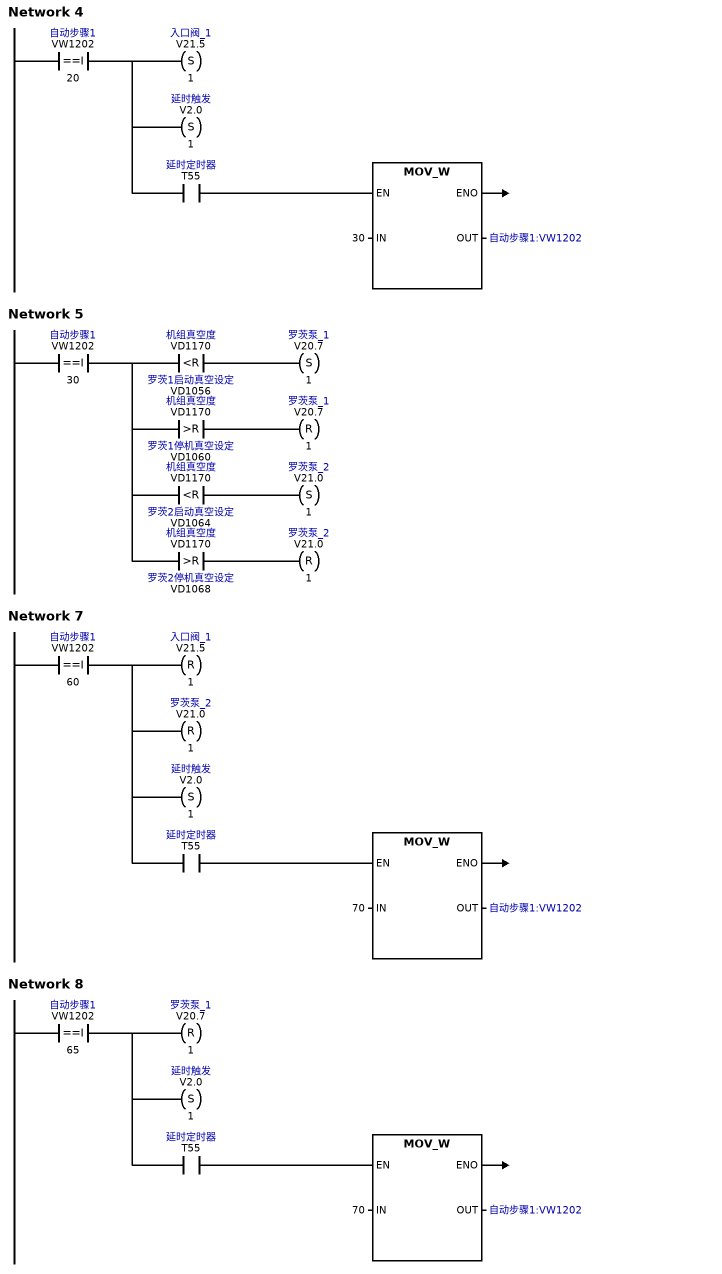
Network 4
LDW=   自动步骤1:VW1202, 20
S      入口阀_1:V21.5, 1
S      延时触发:V2.0, 1
A      延时定时器:T55
MOVW   30, 自动步骤1:VW1202
Network 5
LDW=   自动步骤1:VW1202, 30
LPS
AR<    机组真空度:VD1170, 罗茨1启动真空设定:VD1056
S      罗茨泵_1:V20.7, 1
LRD
AR>    机组真空度:VD1170, 罗茨1停机真空设定:VD1060
R      罗茨泵_1:V20.7, 1
LRD
AR<    机组真空度:VD1170, 罗茨2启动真空设定:VD1064
S      罗茨泵_2:V21.0, 1
LPP
AR>    机组真空度:VD1170, 罗茨2停机真空设定:VD1068
R      罗茨泵_2:V21.0, 1
Network 7
LDW=   自动步骤1:VW1202, 60
R      入口阀_1:V21.5, 1
R      罗茨泵_2:V21.0, 1
S      延时触发:V2.0, 1
A      延时定时器:T55
MOVW   70, 自动步骤1:VW1202
Network 8
LDW=   自动步骤1:VW1202, 65
R      罗茨泵_1:V20.7, 1
S      延时触发:V2.0, 1
A      延时定时器:T55
MOVW   70, 自动步骤1:VW1202
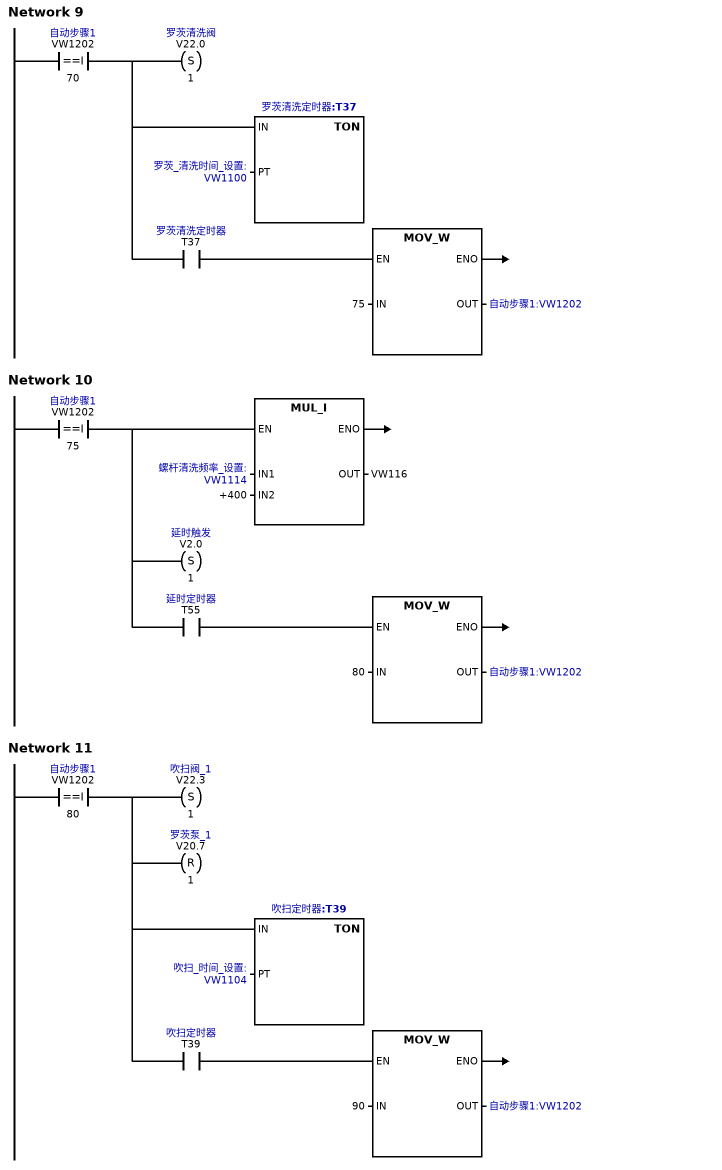
Network 9
LDW=   自动步骤1:VW1202, 70
S      罗茨清洗阀:V22.0, 1
TON    罗茨清洗定时器:T37, 罗茨_清洗时间_设置:VW1100
A      罗茨清洗定时器:T37
MOVW   75, 自动步骤1:VW1202
Network 10
LDW=   自动步骤1:VW1202, 75
MOVW   螺杆清洗频率_设置:VW1114, VW116
*I     +400, VW116
S      延时触发:V2.0, 1
A      延时定时器:T55
MOVW   80, 自动步骤1:VW1202
Network 11
LDW=   自动步骤1:VW1202, 80
S      吹扫阀_1:V22.3, 1
R      罗茨泵_1:V20.7, 1
TON    吹扫定时器:T39, 吹扫_时间_设置:VW1104
A      吹扫定时器:T39
MOVW   90, 自动步骤1:VW1202
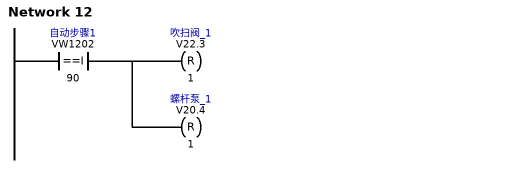
Network 12
LDW=   自动步骤1:VW1202, 90
R      吹扫阀_1:V22.3, 1
R      螺杆泵_1:V20.4, 1
END_SUBROUTINE_BLOCK

SUBROUTINE_BLOCK B_ABB_变频器_MODUBS:SBR7
TITLE=程序注释
BEGIN
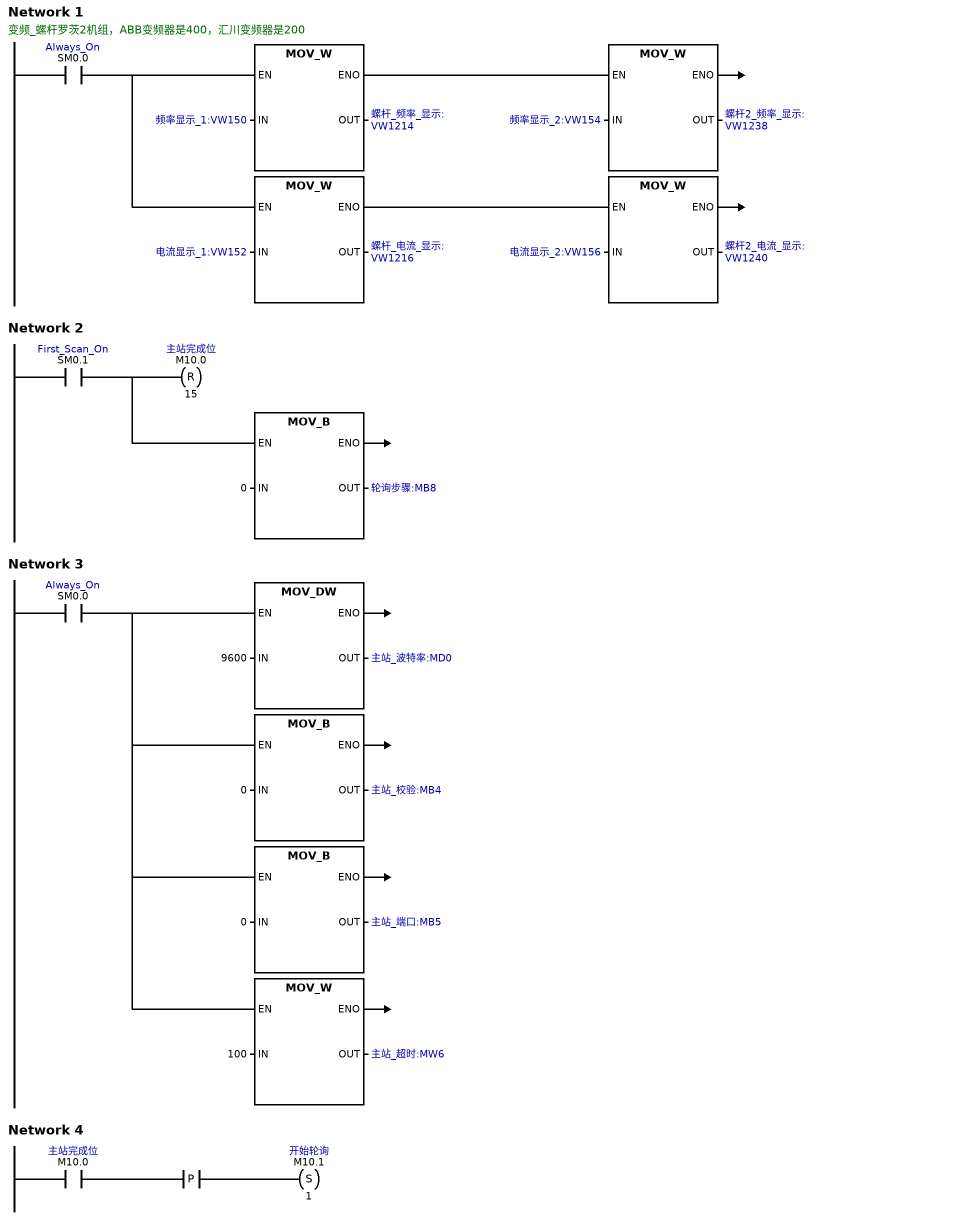
Network 1
// 变频_螺杆罗茨2机组，ABB变频器是400，汇川变频器是200
LD     Always_On:SM0.0
LPS
MOVW   频率显示_1:VW150, 螺杆_频率_显示:VW1214
AENO
MOVW   频率显示_2:VW154, 螺杆2_频率_显示:VW1238
LPP
MOVW   电流显示_1:VW152, 螺杆_电流_显示:VW1216
AENO
MOVW   电流显示_2:VW156, 螺杆2_电流_显示:VW1240
Network 2
LD     First_Scan_On:SM0.1
R      主站完成位:M10.0, 15
MOVB   0, 轮询步骤:MB8
Network 3
LD     Always_On:SM0.0
MOVD   9600, 主站_波特率:MD0
MOVB   0, 主站_校验:MB4
MOVB   0, 主站_端口:MB5
MOVW   100, 主站_超时:MW6
Network 4
LD     主站完成位:M10.0
EU
S      开始轮询:M10.1, 1
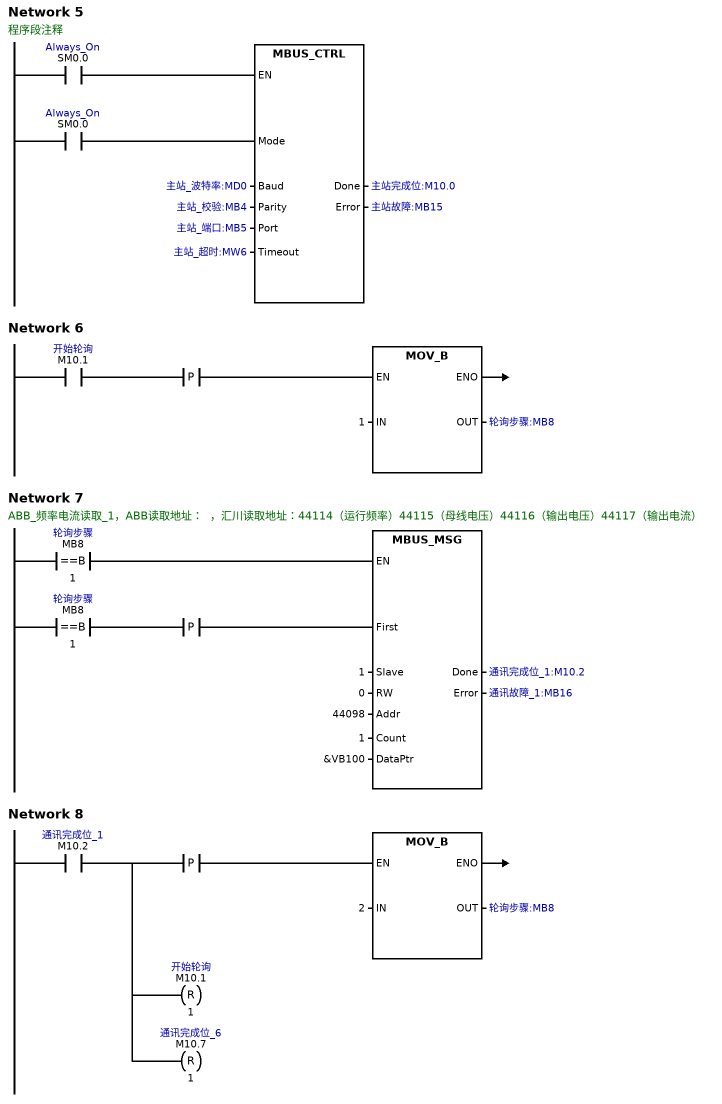
Network 5
// 程序段注释
LD     Always_On:SM0.0
=      L60.0
LD     Always_On:SM0.0
=      L63.7
LD     L60.0
CALL   MBUS_CTRL:SBR8, L63.7, 主站_波特率:MD0, 主站_校验:MB4, 主站_端口:MB5, 主站_超时:MW6, 主站完成位:M10.0, 主站故障:MB15
Network 6
LD     开始轮询:M10.1
EU
MOVB   1, 轮询步骤:MB8
Network 7
// ABB_频率电流读取_1，ABB读取地址：  ，汇川读取地址：44114（运行频率）44115（母线电压）44116（输出电压）44117（输出电流）
LDB=   轮询步骤:MB8, 1
=      L60.0
LDB=   轮询步骤:MB8, 1
EU
=      L63.7
LD     L60.0
CALL   MBUS_MSG:SBR9, L63.7, 1, 0, 44098, 1, &VB100, 通讯完成位_1:M10.2, 通讯故障_1:MB16
Network 8
LD     通讯完成位_1:M10.2
LPS
EU
MOVB   2, 轮询步骤:MB8
LRD
R      开始轮询:M10.1, 1
LPP
R      通讯完成位_6:M10.7, 1
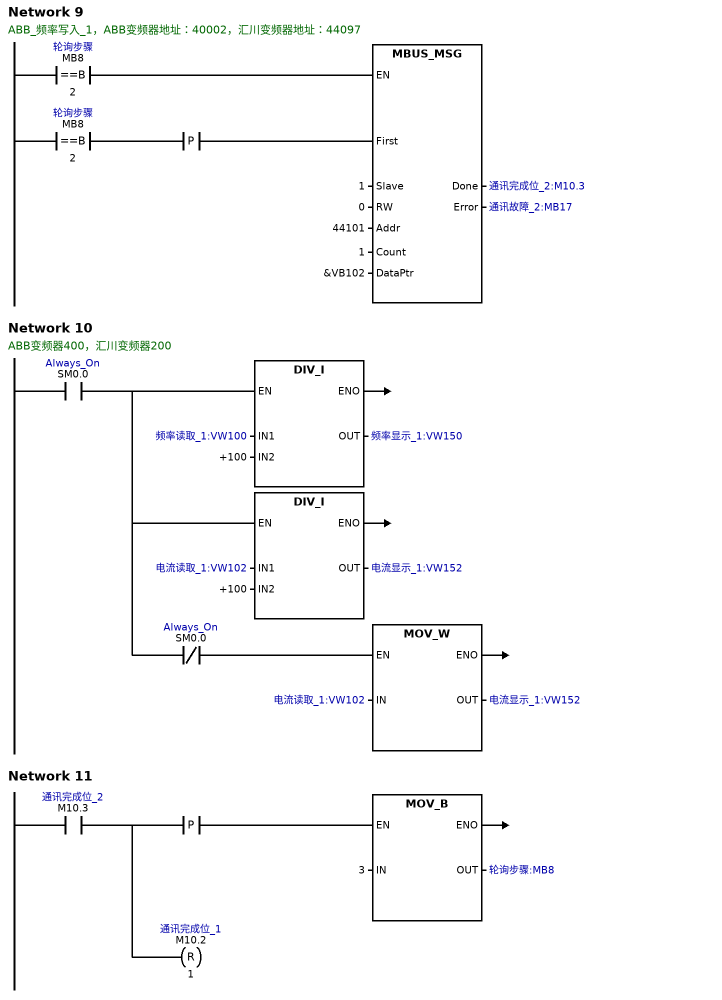
Network 9
// ABB_频率写入_1，ABB变频器地址：40002，汇川变频器地址：44097
LDB=   轮询步骤:MB8, 2
=      L60.0
LDB=   轮询步骤:MB8, 2
EU
=      L63.7
LD     L60.0
CALL   MBUS_MSG:SBR9, L63.7, 1, 0, 44101, 1, &VB102, 通讯完成位_2:M10.3, 通讯故障_2:MB17
Network 10
// ABB变频器400，汇川变频器200
LD     Always_On:SM0.0
MOVW   频率读取_1:VW100, 频率显示_1:VW150
/I     +100, 频率显示_1:VW150
MOVW   电流读取_1:VW102, 电流显示_1:VW152
/I     +100, 电流显示_1:VW152
AN     Always_On:SM0.0
MOVW   电流读取_1:VW102, 电流显示_1:VW152
Network 11
LD     通讯完成位_2:M10.3
LPS
EU
MOVB   3, 轮询步骤:MB8
LPP
R      通讯完成位_1:M10.2, 1
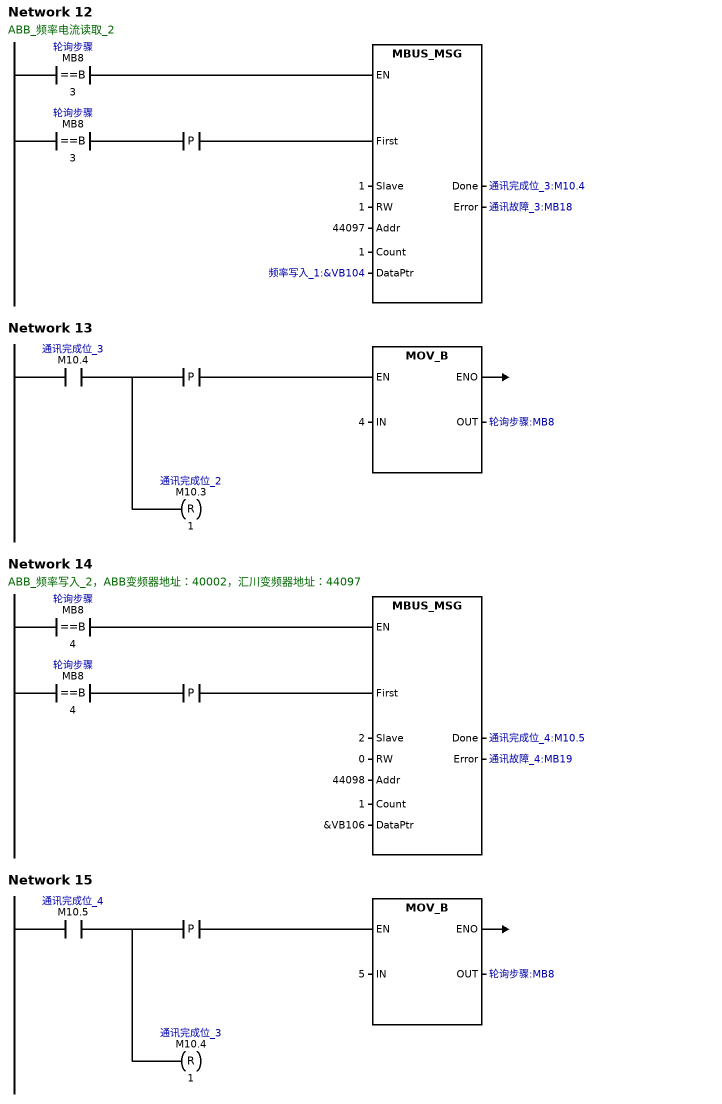
Network 12
// ABB_频率电流读取_2
LDB=   轮询步骤:MB8, 3
=      L60.0
LDB=   轮询步骤:MB8, 3
EU
=      L63.7
LD     L60.0
CALL   MBUS_MSG:SBR9, L63.7, 1, 1, 44097, 1, &频率写入_1:VB104, 通讯完成位_3:M10.4, 通讯故障_3:MB18
Network 13
LD     通讯完成位_3:M10.4
LPS
EU
MOVB   4, 轮询步骤:MB8
LPP
R      通讯完成位_2:M10.3, 1
Network 14
// ABB_频率写入_2，ABB变频器地址：40002，汇川变频器地址：44097
LDB=   轮询步骤:MB8, 4
=      L60.0
LDB=   轮询步骤:MB8, 4
EU
=      L63.7
LD     L60.0
CALL   MBUS_MSG:SBR9, L63.7, 2, 0, 44098, 1, &VB106, 通讯完成位_4:M10.5, 通讯故障_4:MB19
Network 15
LD     通讯完成位_4:M10.5
LPS
EU
MOVB   5, 轮询步骤:MB8
LPP
R      通讯完成位_3:M10.4, 1
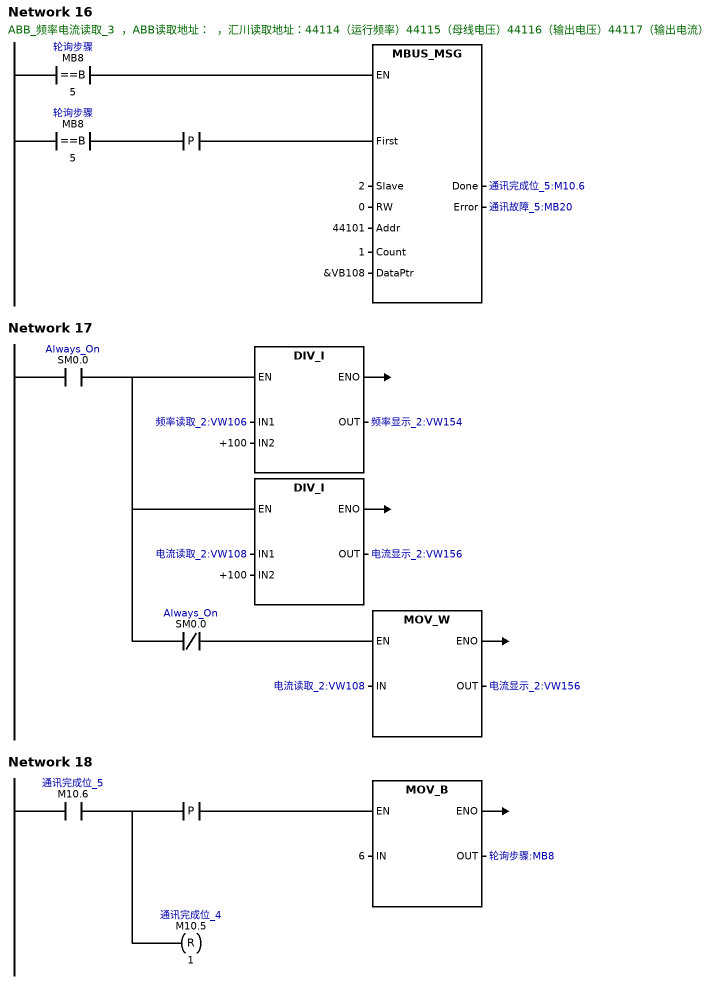
Network 16
// ABB_频率电流读取_3  ，ABB读取地址：  ，汇川读取地址：44114（运行频率）44115（母线电压）44116（输出电压）44117（输出电流）
LDB=   轮询步骤:MB8, 5
=      L60.0
LDB=   轮询步骤:MB8, 5
EU
=      L63.7
LD     L60.0
CALL   MBUS_MSG:SBR9, L63.7, 2, 0, 44101, 1, &VB108, 通讯完成位_5:M10.6, 通讯故障_5:MB20
Network 17
LD     Always_On:SM0.0
MOVW   频率读取_2:VW106, 频率显示_2:VW154
/I     +100, 频率显示_2:VW154
MOVW   电流读取_2:VW108, 电流显示_2:VW156
/I     +100, 电流显示_2:VW156
AN     Always_On:SM0.0
MOVW   电流读取_2:VW108, 电流显示_2:VW156
Network 18
LD     通讯完成位_5:M10.6
LPS
EU
MOVB   6, 轮询步骤:MB8
LPP
R      通讯完成位_4:M10.5, 1
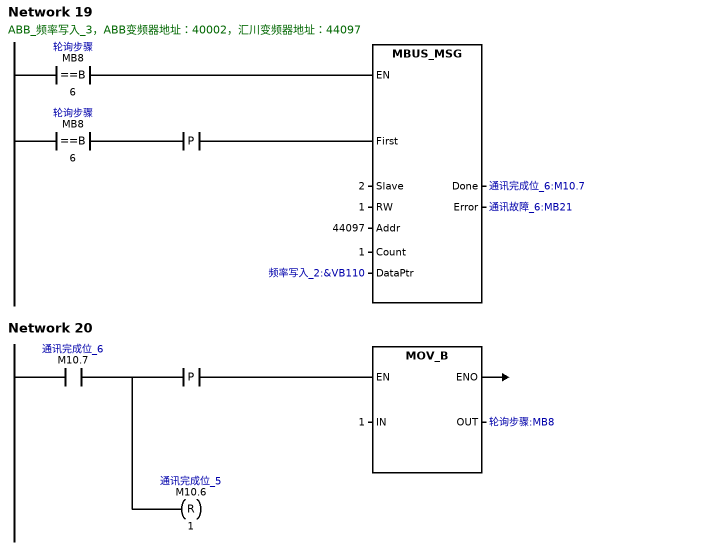
Network 19
// ABB_频率写入_3，ABB变频器地址：40002，汇川变频器地址：44097
LDB=   轮询步骤:MB8, 6
=      L60.0
LDB=   轮询步骤:MB8, 6
EU
=      L63.7
LD     L60.0
CALL   MBUS_MSG:SBR9, L63.7, 2, 1, 44097, 1, &频率写入_2:VB110, 通讯完成位_6:M10.7, 通讯故障_6:MB21
Network 20
LD     通讯完成位_6:M10.7
LPS
EU
MOVB   1, 轮询步骤:MB8
LPP
R      通讯完成位_5:M10.6, 1
Network 28
// 程序段注释
END_SUBROUTINE_BLOCK

// SBR8: protected block, not included

// SBR9: protected block, not included

// SBR10: protected block, not included

SUBROUTINE_BLOCK A_指令转换:SBR11
TITLE=子程序注释
BEGIN
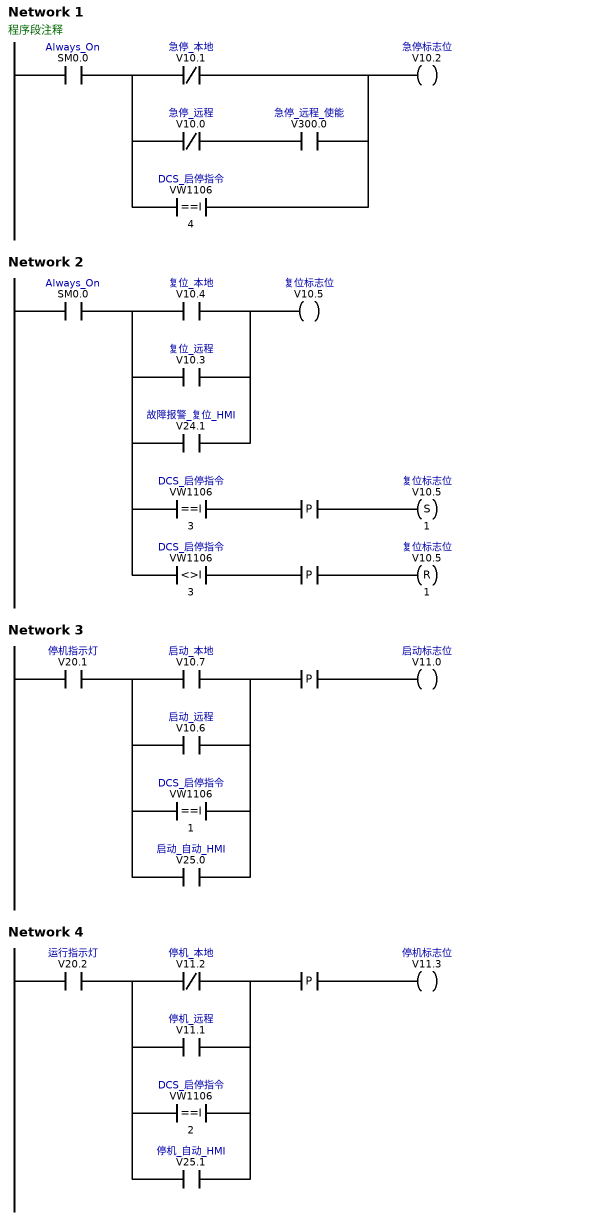
Network 1
// 程序段注释
LD     Always_On:SM0.0
LDN    急停_本地:V10.1
LDN    急停_远程:V10.0
A      急停_远程_使能:V300.0
OLD
OW=    DCS_启停指令:VW1106, 4
ALD
=      急停标志位:V10.2
Network 2
LD     Always_On:SM0.0
LPS
LD     复位_本地:V10.4
O      复位_远程:V10.3
O      故障报警_复位_HMI:V24.1
ALD
=      复位标志位:V10.5
LPP
LPS
AW=    DCS_启停指令:VW1106, 3
EU
S      复位标志位:V10.5, 1
LPP
AW<>   DCS_启停指令:VW1106, 3
EU
R      复位标志位:V10.5, 1
Network 3
LD     停机指示灯:V20.1
LD     启动_本地:V10.7
O      启动_远程:V10.6
OW=    DCS_启停指令:VW1106, 1
O      启动_自动_HMI:V25.0
ALD
EU
=      启动标志位:V11.0
Network 4
LD     运行指示灯:V20.2
LDN    停机_本地:V11.2
O      停机_远程:V11.1
OW=    DCS_启停指令:VW1106, 2
O      停机_自动_HMI:V25.1
ALD
EU
=      停机标志位:V11.3
